PROGRAM MAIN
VAR
END_VAR

END_PROGRAM

(* stored: Version 1.1.0.1
   POU MAIN: Id {c56fa186-ffca-4687-b47f-3aa38dfdad0e} *)
